(* CODESYS project C3FtpClientV1_2_0.project

Project tree, tasks and I/O mapping:
  Device : XV300, Eaton Automation, version 3.5.19.30
    application Application
      libraries: EA23_FtpClient, * (Eaton Automation); Standard, 3.5.18.0 (System)
      task MainTask (cyclic, interval t#10ms, priority 1) calls PLC_PRG
      task FtpTask (cyclic, interval t#100ms, priority 2) calls prgTransfertFTP
      program PLC_PRG [ST]
      program prgTransfertFTP [ST]
      A_lire
  00000000-0000-0000-0000-000000000000|C:\Users\e8000927\Desktop\C3FtpClient\A_lire.pdf
*)

// Device/Application/PLC_PRG
PROGRAM PLC_PRG
VAR
END_VAR

;

END_PROGRAM

// Device/Application/prgTransfertFTP
PROGRAM prgTransfertFTP
VAR
(* Variables generales *)
	dw_Handle	: DWORD;		// ID de la connexion 
	w_ErrorCode	: WORD;			// Code erreur (voir plus bas)
	x_Connected	: BOOL;			// Connecte au serveur

(* Variables d'ouverture *)
	x_Open				: BOOL;
	fb_OpenConnection	: FTP_OpenConnection;
	s_ServerFTP			: STRING(80) := '192.168.1.205';	// Adresse du serveur FTP (Hostname ou adresse IP)
	s_ServerUsername	: STRING(80) := 'User';				// Laisser vide si connexion "anonyme"
	s_ServerPassword	: STRING(80) := 'Password';			// Laisser vide si connexion "anonyme"

(* Variables d'exploration *)
	x_ReadDirectory 		: BOOL;					
	fb_ReadDirectory		: FTP_ReadDirectory;
	s_ReadDirectoryEntry 	: STRING;				// Chemin du repertoire a explorer
	w_DirectoryEntryCount 	: WORD;					// Nombre de fichiers dans le repertoire

(* Variables de transfert de fichiers *)
	x_GetFile	: BOOL;
	fb_GetFile	: FTP_GetFile;
	
	x_PutFile	: BOOL;
	fb_PutFile	: FTP_PutFile;

	s_ServerFile: STRING := 'test4.txt';					// Nom du fichier sur le serveur
	s_PlcFile	: STRING := '/InternalStorage/test4.txt';	// Emplacement et nom du fichier sur l'automate
	
(* Variables de fermeture *)
	x_Close		: BOOL;
	
END_VAR

(* == Table d'aide ================================================================================	*)
(*																									*)
(*	1	FTP_NO_HOST_NAME				Adresse de serveur non definie								*)
(*	2	FTP_CONNECT_ERROR				La connexion avec le serveur n'a pas pu etre etablie		*)
(*	3	FTP_WRONG_HANDLE				Mauvais handle												*)
(*	4	FTP_NO_FILE_ADDRESS				Nom de fichier non defini									*)
(*	5	FTP_GET_FILE_ERROR				Le fichier ne peut pas etre lu								*)
(*	6	FTP_PUT_FILE_ERROR				Le fichier ne peut pas etre ecrit							*)
(*	7	FTP_CHANGE_DIR_ERROR			Le repertoire ne peux etre change							*)
(*	8	FTP_FIND_FIRST_FILE				Le premier repertoire ne peut pas etre lu					*)
(*	9	FTP_FIND_NEXT_FILE				Le repertoire suivant ne peut pas etre lu					*)
(*	10	FTP_DELETE_FILE_ERROR			Le ficchier ne peut pas etre efface							*)
(*	11	FTP_TO_MANY_OPEN_CONNECTION		Trop de connexions ouvertes (MAX. 100)						*)
(* ================================================================================================	*)

(*=================================================================================================
	Programme exemple de client FTP
===================================================================================================
	Nom :		C3FtpClient
	Date :		18/07/2024
	Version :	V1.2.0
	Materiel :	XV300
	CoDeSys :	V3.5.19.30
	Auteur :	Bruno COTTANCIN
	Libs :		EA23_FtpClient.library
===================================================================================================
	NOTE IMPORTANTE !
	~~~~~~~~~~~~~~~
		Nous vous rappellons que ceci est un exemple de programme dont l’objectif est de vérifier
		le bon fonctionnement de l’application.
		Vous pouvez utiliser cet exemple de programme mais nous vous conseillons de tester son
		fonctionnement dans des conditions qui NE mettront pas l’installation en péril.
		La mise en œuvre et l’exploitation de ce programme sont sous votre responsabilité.
===================================================================================================
	Versions
		- V1.1.0		Version originale											(18/01/2018)	
		- V1.2.0		Mise a jour des bibliotheques et version XV300				(18/07/2024)	
		
=================================================================================================*)



(* === Ouverture de la connexion FTP =========================================================== *)
IF x_Open THEN
	x_Open := FALSE;
	fb_OpenConnection(
		psHost		:= ADR (s_ServerFTP), 
		psUsername	:= ADR (s_ServerUsername), 
		psPassword	:= ADR (s_ServerPassword), 
		hFtpOpen	=> dw_Handle,
		xError 		=> , 
		wErrorId	=> w_ErrorCode
	);
	IF fb_OpenConnection.xError THEN
		(* Gestion de l'erreur *)
		x_Connected := FALSE;
	ELSE
		x_Connected := TRUE;
	END_IF;
END_IF;


(* === Exploration du repertoire =============================================================== *)
IF x_ReadDirectory THEN
	x_ReadDirectory := FALSE;
	w_DirectoryEntryCount := 0;
	REPEAT												// Repeter tant qu'il y a des fichiers
		fb_ReadDirectory (
			hFtpOpen 			:= dw_Handle,
			psDirectoryEntry 	:= ADR(s_ReadDirectoryEntry),
			xDirectoryEntry		=> , 
			xDirectory			=> , 
			dwFileSize			=> , 
			xError				=> , 
			wErrorId			=> w_ErrorCode
		);
		IF fb_ReadDirectory.xError THEN
			(* Gestion de l'erreur *)
			EXIT;
		ELSE
			IF fb_ReadDirectory.xDirectoryEntry THEN	// Compteur de fichier
				w_DirectoryEntryCount := w_DirectoryEntryCount + 1;
			END_IF;
		END_IF;
	UNTIL fb_ReadDirectory.xDirectoryEntry = FALSE		// Fin d'exploration
	END_REPEAT;
END_IF;


(* === Transfert de fichier du serveur vers l'automate ========================================= *)
IF x_GetFile THEN
	x_GetFile := FALSE;
	fb_GetFile (
		hFtpOpen 	:= dw_Handle,
		psSrcFile	:= ADR(s_ServerFile),
		psDstFile	:= ADR(s_PlcFile),
		xError		=> ,
		wErrorId	=> w_ErrorCode
	);
	IF fb_GetFile.xError THEN
		(* Gestion de l'erreur *)
	END_IF;
END_IF;


(* === Transfert de fichier de l'automate vers le serveur ====================================== *)
IF x_PutFile THEN
	x_PutFile := FALSE;
	fb_PutFile(
		hFtpOpen	:= dw_Handle, 
		psSrcFile	:= ADR(s_PlcFile), 
		psDstFile	:= ADR(s_ServerFile), 
		xError		=> , 
		wErrorId	=> w_ErrorCode
	);
	IF fb_PutFile.xError THEN
		(* Gestion de l'erreur *)
	END_IF;
END_IF;


(* === Fermeture de la connexion FTP =========================================================== *)
IF x_Close THEN
	x_Close := FALSE;
	IF NOT FTP_CloseConnection(dw_Handle) THEN
		(* Gestion de l'erreur *)
	ELSE
		IF x_Connected THEN
			x_Connected := FALSE;
		END_IF;
	END_IF;
END_IF;

END_PROGRAM
